FUNCTION_BLOCK FB_BoxControl
VAR_INPUT
	iMaxNumLimit:USINT:=4;
	
END_VAR
VAR_OUTPUT
END_VAR
VAR
END_VAR
VAR_IN_OUT
		iqBoxdata:structBoxData;
END_VAR
VAR // added by the converter: edge detectors and wires of the graphical bodies
    _rt1, _rt2, _rt3, _rt4 : R_TRIG;
    _w1, _w2, _w3, _w4 : BOOL;
END_VAR

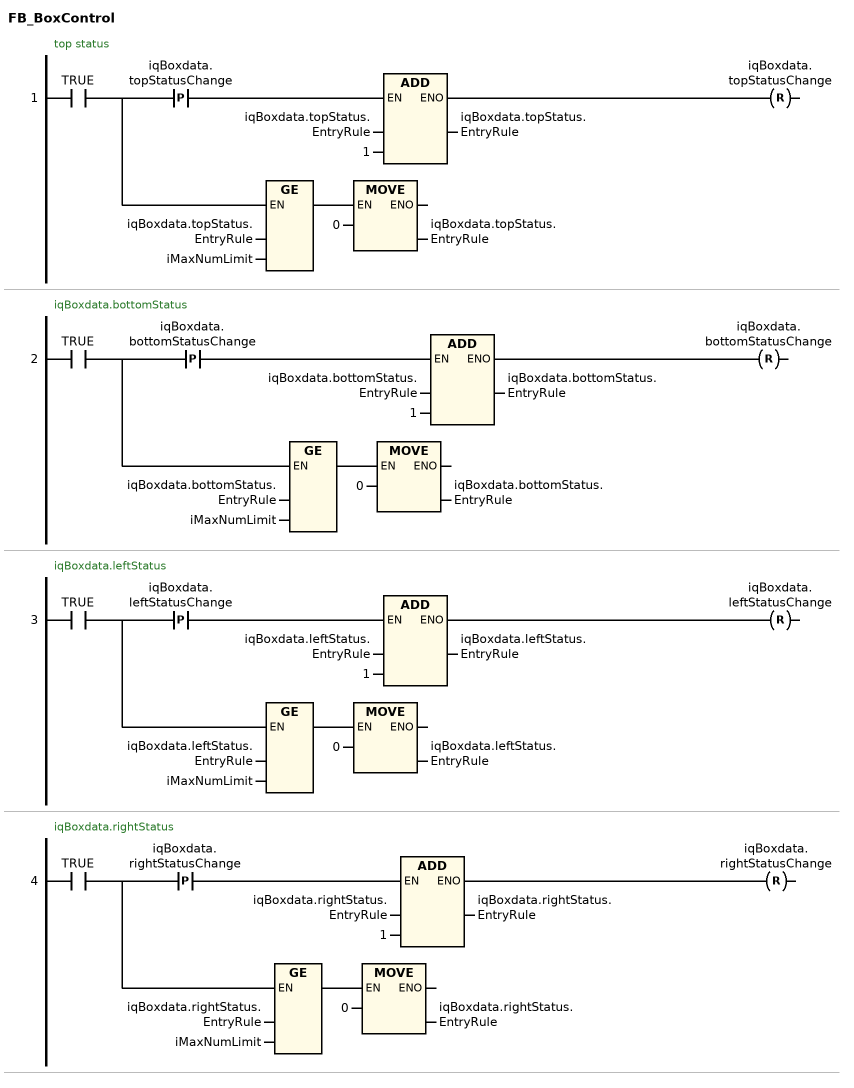
// NETWORK 1
// top status
_rt1(CLK := iqBoxdata.topStatusChange);
_w1 := TRUE AND _rt1.Q;
IF _w1 THEN iqBoxdata.topStatus.EntryRule := iqBoxdata.topStatus.EntryRule + 1; END_IF
iqBoxdata.topStatusChange R= _w1;
IF iqBoxdata.topStatus.EntryRule >= iMaxNumLimit THEN iqBoxdata.topStatus.EntryRule := 0; END_IF

// NETWORK 2
// iqBoxdata.bottomStatus
_rt2(CLK := iqBoxdata.bottomStatusChange);
_w2 := TRUE AND _rt2.Q;
IF _w2 THEN iqBoxdata.bottomStatus.EntryRule := iqBoxdata.bottomStatus.EntryRule + 1; END_IF
iqBoxdata.bottomStatusChange R= _w2;
IF iqBoxdata.bottomStatus.EntryRule >= iMaxNumLimit THEN iqBoxdata.bottomStatus.EntryRule := 0; END_IF

// NETWORK 3
// iqBoxdata.leftStatus
_rt3(CLK := iqBoxdata.leftStatusChange);
_w3 := TRUE AND _rt3.Q;
IF _w3 THEN iqBoxdata.leftStatus.EntryRule := iqBoxdata.leftStatus.EntryRule + 1; END_IF
iqBoxdata.leftStatusChange R= _w3;
IF iqBoxdata.leftStatus.EntryRule >= iMaxNumLimit THEN iqBoxdata.leftStatus.EntryRule := 0; END_IF

// NETWORK 4
// iqBoxdata.rightStatus
_rt4(CLK := iqBoxdata.rightStatusChange);
_w4 := TRUE AND _rt4.Q;
IF _w4 THEN iqBoxdata.rightStatus.EntryRule := iqBoxdata.rightStatus.EntryRule + 1; END_IF
iqBoxdata.rightStatusChange R= _w4;
IF iqBoxdata.rightStatus.EntryRule >= iMaxNumLimit THEN iqBoxdata.rightStatus.EntryRule := 0; END_IF

END_FUNCTION_BLOCK

(* stored: Version 1.1.0.1, ProductVersion 3.1.4024.11
   POU FB_BoxControl: Id {2b5b0c30-c34a-082d-3af5-2acd0c6d64aa}, SpecialFunc None *)
